{attribute 'linkalways'} 
{attribute 'no_explicit_call' := 'This FB is a CLASS and must be accessed using methods or properties'}
{attribute 'enable_dynamic_creation'}
FUNCTION_BLOCK Node_F_VN_MinImageWithScalar EXTENDS VisionNode
VAR
    fScalar : _LREAL(0.0);
    ipSrcImage : _ITcVnImage;
    ipDestImage : _ITcVnImage;
    hrPrev : _HRESULT(S_OK);
	hresult : _HRESULT(S_OK);
END_VAR

METHOD PUBLIC  Clone : I_Node
VAR
	pNode : POINTER TO Node_F_VN_MinImageWithScalar;
END_VAR
pNode := __NEW(Node_F_VN_MinImageWithScalar);
Clone := pNode^;
END_METHOD

METHOD FB_init : BOOL
VAR_INPUT
	bInitRetains : BOOL; // if TRUE, the retain variables are initialized (warm start / cold start)
	bInCopyCode : BOOL;  // if TRUE, the instance afterwards gets moved into the copy code (online change)
END_VAR
AddInput('fScalar', fScalar);
AddInput('ipSrcImage', ipSrcImage);
AddInput('hrPrev', hrPrev);
AddOutput('ipDestImage', ipDestImage);
AddOutput('hresult',hresult);
END_METHOD

METHOD PROTECTED OnExecute
hresult.Value := F_VN_MinImageWithScalar(
    fScalar := fScalar.Value,
    ipSrcImage := ipSrcImage.Value,
	ipDestImage := ipDestImage.Value,
	hrPrev:= hrPrev.Value);
END_METHOD

METHOD PUBLIC PreExecutionCheck
VAR_INPUT
	Check : I_PreExecutionChecks;
END_VAR
Check.IsTrue(ipSrcImage.IsValid, 'ipSrcImage must contain an image');
END_METHOD

END_FUNCTION_BLOCK

(* stored: Version 1.1.0.1, ProductVersion 3.1.4024.13
   POU Node_F_VN_MinImageWithScalar: Id {c345d6f5-4b36-07ed-3bcf-1f6f682c772a}, SpecialFunc None
   Folder Constructor: Id {3b61f6ba-9f8b-0329-0d87-51e1243bb889}
   Method Clone: Id {8cf8b137-2416-0773-1041-05c2a7b1140f}
   Method FB_init: Id {2c6e5b64-7782-0e93-27e5-0cae6b554626}
   Method OnExecute: Id {4f46db6f-2406-0ca0-0d77-1539ec2dd097}
   Method PreExecutionCheck: Id {e0c860e6-f1f7-0699-3a9f-fad8c6490821} *)
